{attribute 'GeneratedUsingTerminal: KL6211-0002'}
{attribute addProperty BoxType "KL6211-0002"}
{attribute addProperty Id "StatusAT %I*UINT0Parameter_InAT %I*UDINT0ASI_In_Slave_1_StatusAT %I*USINT0ASI_In_Slave_3_Slave_2AT %I*USINT0ASI_In_Slave_5_Slave_4AT %I*USINT0ASI_In_Slave_7_Slave_6AT %I*USINT0ASI_In_Slave_9_Slave_8AT %I*USINT0ASI_In_Slave_11_Slave_10AT %I*USINT0ASI_In_Slave_13_Slave_12AT %I*USINT0ASI_In_Slave_15_Slave_14AT %I*USINT0ASI_In_Slave_17_Slave_16AT %I*USINT0ASI_In_Slave_19_Slave_18AT %I*USINT0ASI_In_Slave_21_Slave_20AT %I*USINT0ASI_In_Slave_23_Slave_22AT %I*USINT0ASI_In_Slave_25_Slave_24AT %I*USINT0ASI_In_Slave_27_Slave_26AT %I*USINT0ASI_In_Slave_29_Slave_28AT %I*USINT0ASI_In_Slave_31_Slave_30AT %I*USINT0ControlAT %Q*UINT0Parameter_OutAT %Q*UDINT0ASI_Out_Slave_1_ControlAT %Q*USINT0ASI_Out_Slave_3_Slave_2AT %Q*USINT0ASI_Out_Slave_5_Slave_4AT %Q*USINT0ASI_Out_Slave_7_Slave_6AT %Q*USINT0ASI_Out_Slave_9_Slave_8AT %Q*USINT0ASI_Out_Slave_11_Slave_10AT %Q*USINT0ASI_Out_Slave_13_Slave_12AT %Q*USINT0ASI_Out_Slave_15_Slave_14AT %Q*USINT0ASI_Out_Slave_17_Slave_16AT %Q*USINT0ASI_Out_Slave_19_Slave_18AT %Q*USINT0ASI_Out_Slave_21_Slave_20AT %Q*USINT0ASI_Out_Slave_23_Slave_22AT %Q*USINT0ASI_Out_Slave_25_Slave_24AT %Q*USINT0ASI_Out_Slave_27_Slave_26AT %Q*USINT0ASI_Out_Slave_29_Slave_28AT %Q*USINT0ASI_Out_Slave_31_Slave_30AT %Q*USINT0"}
{attribute addProperty CRC "2192429174"}
{attribute addProperty Size "0"}
TYPE Channel_82ADD076 :
STRUCT
	{attribute addProperty Name "Status"}
	Status AT %I* : UINT;
	{attribute addProperty Name "Parameter_In"}
	Parameter_In AT %I* : UDINT;
	{attribute addProperty Name "ASI_In_Slave_1_Status"}
	ASI_In_Slave_1_Status AT %I* : USINT;
	{attribute addProperty Name "ASI_In_Slave_3_Slave_2"}
	ASI_In_Slave_3_Slave_2 AT %I* : USINT;
	{attribute addProperty Name "ASI_In_Slave_5_Slave_4"}
	ASI_In_Slave_5_Slave_4 AT %I* : USINT;
	{attribute addProperty Name "ASI_In_Slave_7_Slave_6"}
	ASI_In_Slave_7_Slave_6 AT %I* : USINT;
	{attribute addProperty Name "ASI_In_Slave_9_Slave_8"}
	ASI_In_Slave_9_Slave_8 AT %I* : USINT;
	{attribute addProperty Name "ASI_In_Slave_11_Slave_10"}
	ASI_In_Slave_11_Slave_10 AT %I* : USINT;
	{attribute addProperty Name "ASI_In_Slave_13_Slave_12"}
	ASI_In_Slave_13_Slave_12 AT %I* : USINT;
	{attribute addProperty Name "ASI_In_Slave_15_Slave_14"}
	ASI_In_Slave_15_Slave_14 AT %I* : USINT;
	{attribute addProperty Name "ASI_In_Slave_17_Slave_16"}
	ASI_In_Slave_17_Slave_16 AT %I* : USINT;
	{attribute addProperty Name "ASI_In_Slave_19_Slave_18"}
	ASI_In_Slave_19_Slave_18 AT %I* : USINT;
	{attribute addProperty Name "ASI_In_Slave_21_Slave_20"}
	ASI_In_Slave_21_Slave_20 AT %I* : USINT;
	{attribute addProperty Name "ASI_In_Slave_23_Slave_22"}
	ASI_In_Slave_23_Slave_22 AT %I* : USINT;
	{attribute addProperty Name "ASI_In_Slave_25_Slave_24"}
	ASI_In_Slave_25_Slave_24 AT %I* : USINT;
	{attribute addProperty Name "ASI_In_Slave_27_Slave_26"}
	ASI_In_Slave_27_Slave_26 AT %I* : USINT;
	{attribute addProperty Name "ASI_In_Slave_29_Slave_28"}
	ASI_In_Slave_29_Slave_28 AT %I* : USINT;
	{attribute addProperty Name "ASI_In_Slave_31_Slave_30"}
	ASI_In_Slave_31_Slave_30 AT %I* : USINT;
	{attribute addProperty Name "Control"}
	Control AT %Q* : UINT;
	{attribute addProperty Name "Parameter_Out"}
	Parameter_Out AT %Q* : UDINT;
	{attribute addProperty Name "ASI_Out_Slave_1_Control"}
	ASI_Out_Slave_1_Control AT %Q* : USINT;
	{attribute addProperty Name "ASI_Out_Slave_3_Slave_2"}
	ASI_Out_Slave_3_Slave_2 AT %Q* : USINT;
	{attribute addProperty Name "ASI_Out_Slave_5_Slave_4"}
	ASI_Out_Slave_5_Slave_4 AT %Q* : USINT;
	{attribute addProperty Name "ASI_Out_Slave_7_Slave_6"}
	ASI_Out_Slave_7_Slave_6 AT %Q* : USINT;
	{attribute addProperty Name "ASI_Out_Slave_9_Slave_8"}
	ASI_Out_Slave_9_Slave_8 AT %Q* : USINT;
	{attribute addProperty Name "ASI_Out_Slave_11_Slave_10"}
	ASI_Out_Slave_11_Slave_10 AT %Q* : USINT;
	{attribute addProperty Name "ASI_Out_Slave_13_Slave_12"}
	ASI_Out_Slave_13_Slave_12 AT %Q* : USINT;
	{attribute addProperty Name "ASI_Out_Slave_15_Slave_14"}
	ASI_Out_Slave_15_Slave_14 AT %Q* : USINT;
	{attribute addProperty Name "ASI_Out_Slave_17_Slave_16"}
	ASI_Out_Slave_17_Slave_16 AT %Q* : USINT;
	{attribute addProperty Name "ASI_Out_Slave_19_Slave_18"}
	ASI_Out_Slave_19_Slave_18 AT %Q* : USINT;
	{attribute addProperty Name "ASI_Out_Slave_21_Slave_20"}
	ASI_Out_Slave_21_Slave_20 AT %Q* : USINT;
	{attribute addProperty Name "ASI_Out_Slave_23_Slave_22"}
	ASI_Out_Slave_23_Slave_22 AT %Q* : USINT;
	{attribute addProperty Name "ASI_Out_Slave_25_Slave_24"}
	ASI_Out_Slave_25_Slave_24 AT %Q* : USINT;
	{attribute addProperty Name "ASI_Out_Slave_27_Slave_26"}
	ASI_Out_Slave_27_Slave_26 AT %Q* : USINT;
	{attribute addProperty Name "ASI_Out_Slave_29_Slave_28"}
	ASI_Out_Slave_29_Slave_28 AT %Q* : USINT;
	{attribute addProperty Name "ASI_Out_Slave_31_Slave_30"}
	ASI_Out_Slave_31_Slave_30 AT %Q* : USINT;
END_STRUCT
END_TYPE

(* stored: Version 1.2.0.0, ProductVersion 3.1.4024.9
   DUT Channel_82ADD076: Id {e8b8e181-8ee7-4bcc-a5c6-4f36712a8fed} *)
